(* PLC project Untitled1, Eclipse Foundation CIF to Structured Text 0.0 *)
(* stored: creationDateTime 1970-01-01T01:00:00 *)

TYPE STATE : STRUCT
  curTime : LREAL;
  dvar_M_p AT %Q* : enum_E;
END_STRUCT;
END_TYPE

TYPE enum_E : (elit_X);
END_TYPE

FUNCTION alg_x : LREAL
  VAR_INPUT
    state : STATE;
  END_VAR

            alg_x := state.curTime;
          
END_FUNCTION

FUNCTION alg_g_a_x : LREAL
  VAR_INPUT
    state : STATE;
  END_VAR

            alg_g_a_x := state.curTime;
          
END_FUNCTION

FUNCTION alg_g_z : LREAL
  VAR_INPUT
    state : STATE;
  END_VAR

            alg_g_z := state.curTime;
          
END_FUNCTION

FUNCTION alg_g_z2 : LREAL
  VAR_INPUT
    state : STATE;
  END_VAR

            alg_g_z2 := state.curTime;
          
END_FUNCTION

FUNCTION alg_g_w_w : LREAL
  VAR_INPUT
    state : STATE;
  END_VAR

            alg_g_w_w := state.curTime;
          
END_FUNCTION

FUNCTION alg_g_w_W2 : LREAL
  VAR_INPUT
    state : STATE;
  END_VAR

            alg_g_w_W2 := state.curTime;
          
END_FUNCTION

FUNCTION alg_g_a_X2 : LREAL
  VAR_INPUT
    state : STATE;
  END_VAR

            alg_g_a_X2 := state.curTime;
          
END_FUNCTION

PROGRAM MAIN
  VAR_OUTPUT
    timerValue0 : TIME;
    timerValue1 : TIME;
  END_VAR
  VAR
    cnt : LINT;
    first : BOOL := TRUE;
    curTimerValue : TIME;
    state0 : STATE;
    curTime : LREAL;
    loopsKilled : LINT;
  END_VAR
  VAR_TEMP
    lastTimerValue : TIME;
    curDeltaTime : TIME;
    curDeltaSecs : LREAL;
    state1 : STATE;
    progress : BOOL;
    loopCount : INT;
  END_VAR

            
// Handle 'time' and cycle time.
cnt := cnt + 1;

timer0(IN := curTimer = 0, PT := T#1D);
timer1(IN := curTimer = 1, PT := T#1D);
timerValue0 := timer0.ET;
timerValue1 := timer1.ET;

lastTimerValue := curTimerValue;
IF curTimer = 0 THEN
    curTimerValue := timerValue0;
ELSE
    curTimerValue := timerValue1;
END_IF;
curDeltaTime := curTimerValue - lastTimerValue;
curDeltaSecs := TIME_TO_LREAL(curDeltaTime) / 1000;
curTime := curTime + curDeltaSecs;

IF cnt MOD 10 = 0 THEN
    curTimer := 1 - curTimer;
    curTimerValue := T#0S;
    timer0(IN := curTimer = 0, PT := T#1D);
    timer1(IN := curTimer = 1, PT := T#1D);
    timerValue0 := timer0.ET;
    timerValue1 := timer1.ET;
END_IF;

IF first THEN
    first := FALSE;

    // Initialize state variables for initial state.
    state0.dvar_M_p := elit_X;
ELSE
    // Update continuous variables for time delay.

    state0.curTime := curTime;
END_IF;

// Event loop.
WHILE TRUE DO
    progress := FALSE;

    // Done with events?
    IF NOT progress THEN
        EXIT;
    END_IF;

    // Protect against events that are always enabled.
    loopCount := loopCount + 1;
    IF loopCount >= 100 THEN
        loopsKilled := loopsKilled + 1;
        EXIT;
    END_IF;
END_WHILE;
          
END_PROGRAM

CONFIGURATION Untitled1
  RESOURCE Untitled1 ON PLC
    VAR_GLOBAL  (* TIMERS *)
      timer0 : TON;
      timer1 : TON;
      curTimer : INT := 0;
    END_VAR
    TASK PlcTask(INTERVAL := t#10ms, PRIORITY := 20);
    PROGRAM MAIN WITH PlcTask : MAIN;
  END_RESOURCE
END_CONFIGURATION
